Universal Robots PolyScope program: test_gripper.urp

Program test_gripper (installation=default directory=/programs createdIn=5.11.9.1010452 lastSavedIn=5.11.9.1010452 robotSerialNumber=20225200364)
Calibrated DH parameters: a=[0.00002, -0.569483, -0.54992, -0.00001, -0.000036, 0]; d=[0.180894, -146.691669, 192.918669, -46.053088, 0.119778, 0.115602]; alpha=[1.571425, -0.001534, 0.003359, 1.568739, -1.571477, 0]; deltaTheta=[0, 0.376258, -0.101074, -0.275185, -0.000002, 0]
Robot Program (runOnlyOnce=false)
  URCap RG Grip (OnRobot, OnRobot A/S) dataModel(rg-target-force=40.0, Variable(key=on_return, variable(name=on_return)))
  MoveJ speed 60 deg/s, acceleration 80 deg/s^2 (useActiveTCP=true) feature=Base
    Waypoint Waypoint_1: TCP in base x=532.214 y=252.425 z=324.895 mm, rx=0.0022 ry=-3.1416 rz=0 rad; joints [42.517, -89.39, -128.798, -51.776, 90.175, 132.475] deg
    URCap RG Grip (OnRobot, OnRobot A/S) dataModel(rg-target-force=40.0)
    URCap RG Grip (OnRobot, OnRobot A/S) dataModel(rg-target-force=40.0)
